{region '#Template'}
	{attribute 'Version' := '5.0.1.0'}
	{attribute 'Tags' := '"LCID": "1031", "Text": "General, Cabinet, Control cabinet"'}
	{attribute 'Tags' := '"LCID": "1033", "Text": "General, Cabinet, Control cabinet"'}
	{attribute 'Using' := '"Type": "Template", "URI": "EC_ID"'}
	{attribute 'Description' := '"LCID": "1031", "Text": "Schaltschrank Ereignisse"'}
	{attribute 'Description' := '"LCID": "1033", "Text": "Control cabinet events"'}
{endregion}
FUNCTION_BLOCK FB_BA_ControlCabinet EXTENDS FB_BA_ControlCabinetBasic
VAR_INPUT CONSTANT
	Fuse01					: FB_BA_SensorBinary;		
	Fuse02					: FB_BA_SensorBinary;	
	Fuse03					: FB_BA_SensorBinary;	
END_VAR

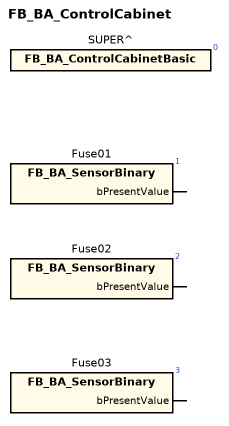
SUPER^(); // FB_BA_ControlCabinetBasic
Fuse01(); // FB_BA_SensorBinary
Fuse02(); // FB_BA_SensorBinary
Fuse03(); // FB_BA_SensorBinary

METHOD FB_init : BOOL
VAR_INPUT
	bInitRetains : BOOL; // if TRUE, the retain variables are initialized (warm start / cold start)
	bInCopyCode : BOOL;  // if TRUE, the instance afterwards gets moved into the copy code (online change)
END_VAR
Fuse01.iParent								:= THIS^;
Fuse01.iLabel								:= LblCtl_Fuse;
Fuse01.sObjectName							:='{Idx=10}';	
Fuse01.eDPADMode							:= E_BA_DPADMode.eInclude;	
Fuse01.Input.iLabel							:= LblFun_Fault;																																									
Fuse01.Input.ePolarity						:= E_BA_Polarity.eReverse;
Fuse01.Input.sActiveText 					:= txtEvent_Triggered;
Fuse01.Input.sInactiveText 					:= txtEvent_Normal;
Fuse01.Input.nEventClassID					:= EC_ID.NC30;
Fuse01.Input.aEventTransitionText[1]		:= txtEvent_Triggered;
Fuse01.Input.aEventTransitionText[2]		:= txtEvent_Error;
Fuse01.Input.aEventTransitionText[3]		:= txtEvent_Normal;
Fuse01.Input.bEventDetectionEnable			:= TRUE;

Fuse01.Input.eEnPlantLock					:= E_BA_LockPriority.eNoLock;	
								 
Fuse02.iParent								:= THIS^;		
Fuse02.iLabel								:= LblCtl_Fuse;	
Fuse02.sObjectName							:='{Idx=20}';	
Fuse02.eDPADMode							:= E_BA_DPADMode.eInclude;	
Fuse02.Input.iLabel							:= LblFun_Fault;																				
Fuse02.Input.ePolarity						:= E_BA_Polarity.eReverse;
Fuse02.Input.sActiveText 					:= txtEvent_Triggered;
Fuse02.Input.sInactiveText 					:= txtEvent_Normal;
Fuse02.Input.nEventClassID					:= EC_ID.NC30;
Fuse02.Input.aEventTransitionText[1]		:= txtEvent_Triggered;
Fuse02.Input.aEventTransitionText[2]		:= txtEvent_Error;
Fuse02.Input.aEventTransitionText[3]		:= txtEvent_Normal;
Fuse02.Input.bEventDetectionEnable			:= TRUE;

Fuse02.Input.eEnPlantLock					:= E_BA_LockPriority.eNoLock;	
										 
Fuse03.iParent								:= THIS^;		
Fuse03.iLabel								:= LblCtl_Fuse;	
Fuse03.sObjectName							:='{Idx=30}';	
Fuse03.eDPADMode							:= E_BA_DPADMode.eInclude;				
Fuse03.Input.iLabel							:= LblFun_Fault;																				
Fuse03.Input.ePolarity						:= E_BA_Polarity.eReverse;
Fuse03.Input.sActiveText 					:= txtEvent_Triggered;
Fuse03.Input.sInactiveText 					:= txtEvent_Normal;
Fuse03.Input.nEventClassID					:= EC_ID.NC30;
Fuse03.Input.aEventTransitionText[1]		:= txtEvent_Triggered;
Fuse03.Input.aEventTransitionText[2]		:= txtEvent_Error;
Fuse03.Input.aEventTransitionText[3]		:= txtEvent_Normal;
Fuse03.Input.bEventDetectionEnable			:= TRUE;

Fuse03.Input.eEnPlantLock					:= E_BA_LockPriority.eNoLock;
END_METHOD

END_FUNCTION_BLOCK

(* stored: Version 1.1.0.1, ProductVersion 3.1.4024.12
   POU FB_BA_ControlCabinet: Id {a79f6a1a-fc45-49e7-80d3-b89bc2dedc88}, SpecialFunc None
   Method FB_init: Id {907425df-4e48-49e5-919a-3e08157b204c} *)
